TYPE ST_MKS_500 EXTENDS ST_VacuumGauge :
STRUCT
	//Discrete Control: Ion gauges only
	i_xHvOn	:	BOOL; //High voltage On to turn on this Cold Cathode gauge
	
	// Simulation parameters
	tonIC	:	TON := (PT := T#10S);// takes 10 seconds to turn on this Cold Cathode gauge
END_STRUCT
END_TYPE

(* stored: Version 1.1.0.1, ProductVersion 3.1.4020.12
   DUT ST_MKS_500: Id {25e9481f-38d0-48ad-928e-1ab5d667df90} *)
